FUNCTION_BLOCK INIT_MQTT_ASYNC
  {SET_ATTRIBUTE(OpcUa, POINT.STARTPOINT)}
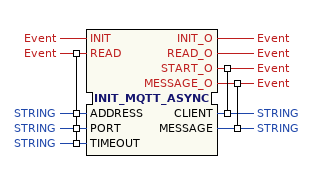
  EVENT_INPUT
    INIT;
    READ WITH ADDRESS, PORT, TIMEOUT;
  END_EVENT
  EVENT_OUTPUT
    INIT_O;
    READ_O;
    START_O WITH CLIENT;
    MESSAGE_O WITH MESSAGE;
  END_EVENT
  VAR_INPUT
    ADDRESS : STRING; {SET_ATTRIBUTE(OpcUa, Constant)}
    PORT : STRING; {SET_ATTRIBUTE(OpcUa, Constant)}
    TIMEOUT : STRING; {SET_ATTRIBUTE(OpcUa, Constant)}
  END_VAR
  VAR_OUTPUT
    CLIENT : STRING; {SET_ATTRIBUTE(OpcUa, Variable)}
    MESSAGE : STRING; {SET_ATTRIBUTE(OpcUa, Variable)}
  END_VAR
END_FUNCTION_BLOCK
